Fanuc KAREL source: KT00783.KL

PROGRAM KT00783
%NOLOCKGROUP
VAR
  S1: STRING[80]
  S2: STRING[80]
  OUT: REAL
BEGIN
  S1 = 'A'
  S2 = 'B'
  S1 = 'A'
  S2 = 'B'
  OUT = ASIN(S1)
END KT00783
